// TIA Portal V17 export
// export: Created 2025-07-17T00:36:36.885756Z, ExportSetting WithDefaults, DisplayName Totally Integrated Automation Portal, DisplayVersion V17, DisplayName TIA Portal Openness, DisplayVersion V17, DisplayName TIA Portal Version Control Interface, DisplayVersion V17, DisplayName STEP 7 Professional, DisplayVersion V17, DisplayName STEP 7 Safety, DisplayVersion V17, DisplayName WinCC Advanced / Unified PC, DisplayVersion V17
ORGANIZATION_BLOCK "Startup"   // OB100, LAD, Startup
TITLE = "Complete Restart"
{ S7_Optimized_Access := 'TRUE' }
VERSION : 0.1
// stored: AutoNumber true, IsIECCheckEnabled false, SetENOAutomatically false
   VAR_INPUT
      LostRetentive : Bool;   // True if retentive data are lost
      LostRTC : Bool;   // True if date and time are lost
   END_VAR
BEGIN

REGION Network 1
   // 建立RS-485连接
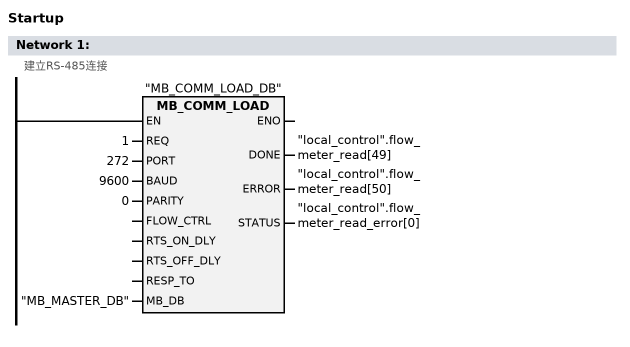
   RUNG wire#powerrail
      "MB_COMM_LOAD_DB".MB_COMM_LOAD(REQ := 1, PORT := 272, BAUD := 9600, PARITY := 0, FLOW_CTRL :=, RTS_ON_DLY :=, RTS_OFF_DLY :=, RESP_TO :=, MB_DB := "MB_MASTER_DB", DONE => "local_control".flow_meter_read[49], ERROR => "local_control".flow_meter_read[50], STATUS => "local_control".flow_meter_read_error[0])
   END_RUNG
   // the same network as SCL:
   "MB_COMM_LOAD_DB"(REQ := 1,   // MB_COMM_LOAD
                     PORT := 272,
                     BAUD := 9600,
                     PARITY := 0,
                     MB_DB := "MB_MASTER_DB",
                     DONE => "local_control".flow_meter_read[49],
                     ERROR => "local_control".flow_meter_read[50],
                     STATUS => "local_control".flow_meter_read_error[0]);
END_REGION
END_ORGANIZATION_BLOCK
